{attribute 'linkalways'} 
{attribute 'no_explicit_call' := 'This FB is a CLASS and must be accessed using methods or properties'}
{attribute 'enable_dynamic_creation'}
FUNCTION_BLOCK InputPortChangedEvent EXTENDS Disposable IMPLEMENTS I_InputPortChangedEvent
VAR
	_target : I_InputPort;
END_VAR

METHOD FB_init : BOOL
VAR_INPUT
	bInitRetains : BOOL; // if TRUE, the retain variables are initialized (warm start / cold start)
	bInCopyCode : BOOL;  // if TRUE, the instance afterwards gets moved into the copy code (online change)
	Target : I_InputPort;
END_VAR
THIS^._target := Target;
END_METHOD

PROPERTY PUBLIC Target : I_InputPort
GET
Target := _target;
END_GET
END_PROPERTY

END_FUNCTION_BLOCK

(* stored: Version 1.1.0.1, ProductVersion 3.1.4024.13
   POU InputPortChangedEvent: Id {0b6e93f0-23d7-45cd-b831-56c837c77c83}, SpecialFunc None
   Folder Constructor: Id {41d7c33b-d71c-4aea-bd39-bdc2e8b2065b}
   Method FB_init: Id {2248bd7c-a96c-410e-a1a8-9ce2844909cc}
   Property Target: Id {6e91ab6d-976b-4bc4-9098-4fcc34dbf993}
   Get Get: Id {ce2fb73c-3af6-4b60-8d3f-7f45e27df121} *)
